// TIA Portal V15.1 export
// export: Created 2024-06-21T08:41:03.9826997Z, ExportSetting WithDefaults, DisplayName Totally Integrated Automation Portal, DisplayVersion V15.1 Update 5, DisplayName TIA Portal Openness, DisplayVersion V15.1 Update 5, DisplayName SINAMICS Startdrive Advanced, DisplayVersion V15.1, DisplayName G130, G150, S120, S150, SINAMICS MV, S210, DisplayVersion V15.1, DisplayName G110M, G120, G120C, G120D, G120P, DisplayVersion V15.1, DisplayName STEP 7 Professional, DisplayVersion V15.1 Update 5, DisplayName STEP 7 Safety, DisplayVersion V15.1, DisplayName WinCC Professional, DisplayVersion V15.1 Update 5, DisplayName SIMATIC Visualization Architect, DisplayVersion V15.1
FUNCTION_BLOCK "LProcTimStrtStop"   // FB1735, FBD
TITLE = LProcTimeStartStop
{ S7_Optimized_Access := 'FALSE' }
AUTHOR : VCC
FAMILY : ProcEq
NAME : TimeStSt
VERSION : 1.0
// ================================================================================
// Module used to give a signal between 2 times with the calendar variable of PLC: 
// start - stop is defined by HMI
// ================================================================================
// stored: AutoNumber false, IsIECCheckEnabled false, SetENOAutomatically False, UDAEnableTagReadback false
   VAR_OUTPUT
      O_TimeActive { ExternalAccessible := 'False'; ExternalVisible := 'False'; ExternalWritable := 'False'} : Bool;   // Time active
      O_InverseTimeActive { ExternalAccessible := 'False'; ExternalVisible := 'False'; ExternalWritable := 'False'} : Bool;   // Inverse Time active
      H_IAnim { ExternalAccessible := 'False'; ExternalVisible := 'False'; ExternalWritable := 'False'} : Word;   // HMI Animation of the icon
   END_VAR
   VAR DB_SPECIFIC
      H_In : Struct   // HMI
         Start : Real := 9.0;   // Start time
         Stop : Real := 9.15;   // Stop time
      END_STRUCT;
      H_Out : Struct   // HMI
         Anim : Word;   // HMI Animation of the object
         DBnr : Int;   // HMI Animation DB number
      END_STRUCT;
      TimeActive { ExternalAccessible := 'False'; ExternalVisible := 'False'; ExternalWritable := 'False'} : Bool;   // Time active
      Start_Int { ExternalAccessible := 'False'; ExternalVisible := 'False'; ExternalWritable := 'False'} : Int := 900;   // Start integer
      Stop_Int { ExternalAccessible := 'False'; ExternalVisible := 'False'; ExternalWritable := 'False'} : Int := 915;   // Stort integer
      DBnr { ExternalAccessible := 'False'; ExternalVisible := 'False'; ExternalWritable := 'False'} : Int;   // HMI DB number
   END_VAR
BEGIN

NETWORK
TITLE = **** 1 - Inputs **** DB number
// DB number
      L     DINO;
      T     #DBnr;

NETWORK
TITLE = **** 4.4 - Machine status - Calculated **** Copy time from HMI to integer
// Copy time from HMI to integer
      L     #H_In.Start;  // Load Start time
      L     100.0;  // * 100
      *R;  // *
      RND;  // Conversion real to integer
      T     #Start_Int;  // Load start time of morning shift = Day 1

      L     #H_In.Stop;  // Load Start time of evening shift - Day 1
      L     100.0;  // * 100
      *R;  // *
      RND;  // Conversion real to integer
      T     #Stop_Int;  // Load start time of evening shift = Day 1


REGION Network 3: **** 4.4 - Machine status - Calculated **** Morning Shift of Day 1
   // Morning Shift of Day 1
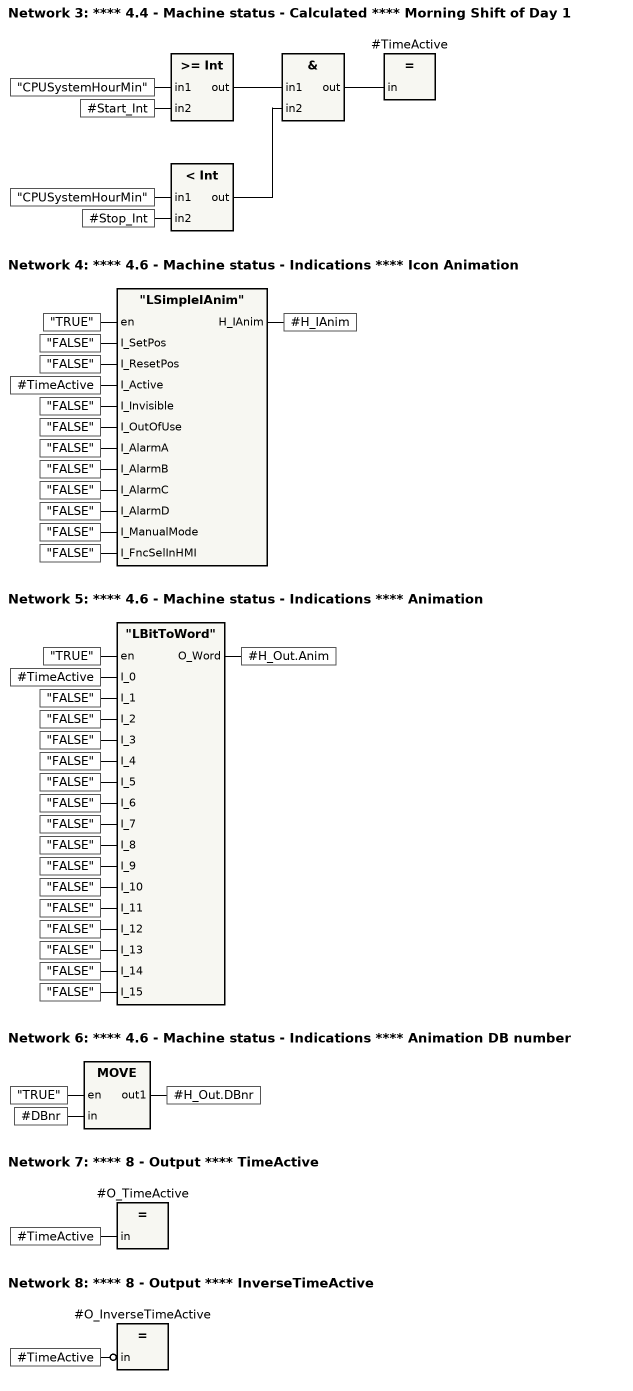
   #TimeActive := ("CPUSystemHourMin" >= #Start_Int) AND ("CPUSystemHourMin" < #Stop_Int);
END_REGION

REGION Network 4: **** 4.6 - Machine status - Indications **** Icon Animation
   // Icon Animation for HMI
   IF "TRUE" THEN
       "LSimpleIAnim"(I_SetPos := "FALSE",
                      I_ResetPos := "FALSE",
                      I_Active := #TimeActive,
                      I_Invisible := "FALSE",
                      I_OutOfUse := "FALSE",
                      I_AlarmA := "FALSE",
                      I_AlarmB := "FALSE",
                      I_AlarmC := "FALSE",
                      I_AlarmD := "FALSE",
                      I_ManualMode := "FALSE",
                      I_FncSelInHMI := "FALSE",
                      H_IAnim => #H_IAnim);
   END_IF;
END_REGION

REGION Network 5: **** 4.6 - Machine status - Indications **** Animation
   // Animation for HMI
   IF "TRUE" THEN
       "LBitToWord"(I_0 := #TimeActive,
                    I_1 := "FALSE",
                    I_2 := "FALSE",
                    I_3 := "FALSE",
                    I_4 := "FALSE",
                    I_5 := "FALSE",
                    I_6 := "FALSE",
                    I_7 := "FALSE",
                    I_8 := "FALSE",
                    I_9 := "FALSE",
                    I_10 := "FALSE",
                    I_11 := "FALSE",
                    I_12 := "FALSE",
                    I_13 := "FALSE",
                    I_14 := "FALSE",
                    I_15 := "FALSE",
                    O_Word => #H_Out.Anim);
   END_IF;
END_REGION

REGION Network 6: **** 4.6 - Machine status - Indications **** Animation DB number
   // Animation DB number
   IF "TRUE" THEN #H_Out.DBnr := #DBnr; END_IF;
END_REGION

REGION Network 7: **** 8 - Output **** TimeActive
   // TimeActive
   #O_TimeActive := #TimeActive;
END_REGION

REGION Network 8: **** 8 - Output **** InverseTimeActive
   // InverseTimeActive
   #O_InverseTimeActive := NOT #TimeActive;
END_REGION
END_FUNCTION_BLOCK
